(* PLC project  *)

PROGRAM P
  VAR
    tmr : TON;
  END_VAR

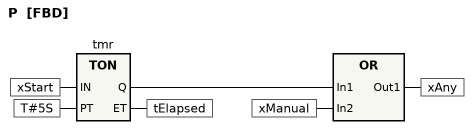
(* FBD diagram, written out as Structured Text *)
tmr(IN := xStart, PT := T#5S);
xAny := tmr.Q OR xManual;
tElapsed := tmr.ET;
END_PROGRAM
